VAR_GLOBAL CONSTANT // CONSTS
    const_d: DINT := 1;
    const_cl: ARRAY[0..2] of LREAL := [1.0, 1.0, 2.0];
    const_x: DINT := -1;
    const_b: DINT := (const_d) + (1);
    const_a: DINT := (const_b) * (2);
    const_c: DINT := (const_a) - (1);
END_VAR

(* stored: ProductVersion 3.1.0.18, Version 1.1.0.1 *)
